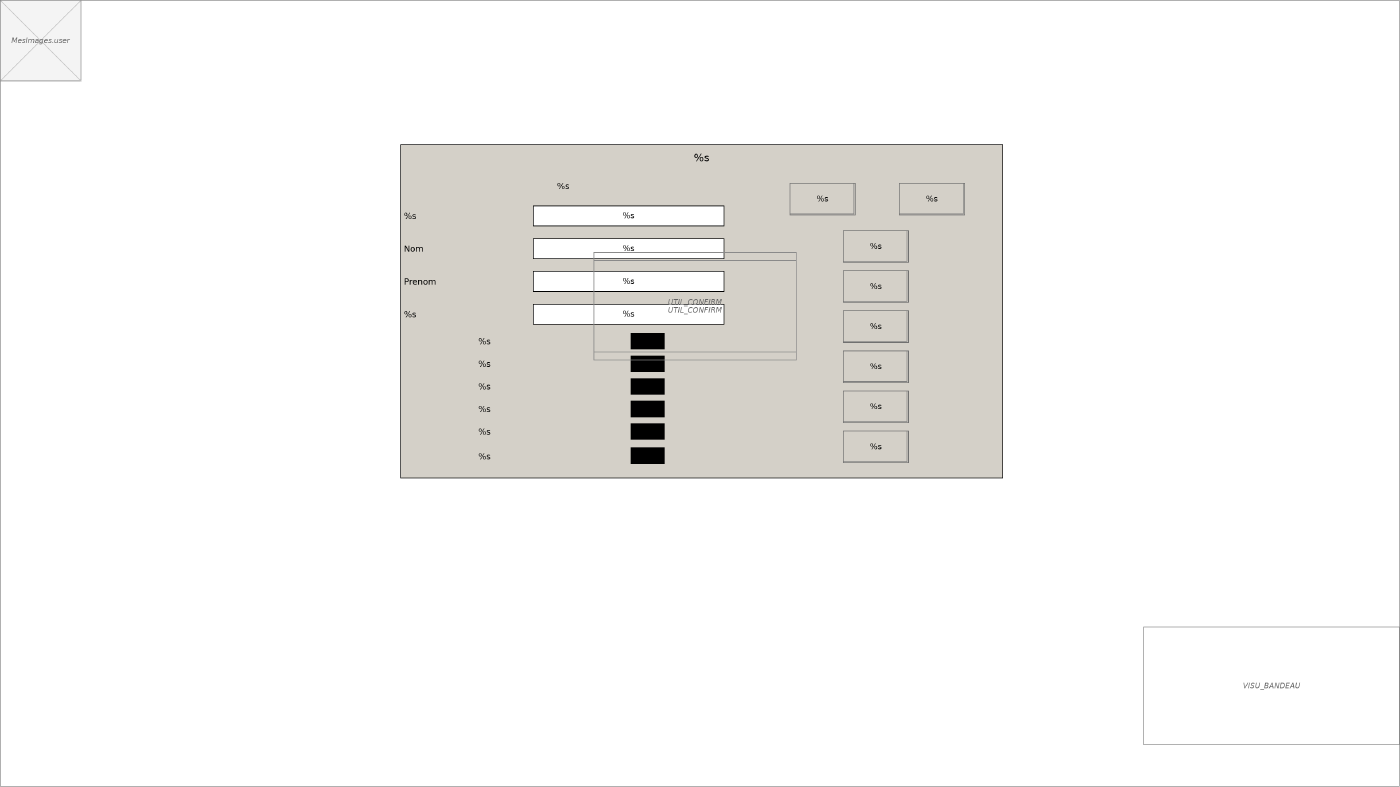
VISUALIZATION UTIL_MENU  // 1920x1080
    Image (0,0 111x111), image: MesImages.user
    RoundedRectangle (549,198 826x458)
    Rectangle (553,202 819x29), "%s", text list: 'TextList_Users_Menu', text index: 1
    Rectangle (731,282 262x28), "%s", text variable: PRG_USER.ACTU_USER.LOGIN
    Rectangle (552,241 441x29), "%s", text list: 'TextList_Users_Menu', text index: 7
    Rectangle (551,282 173x29), "%s", text list: 'TextList_Users_Menu', text index: 5
    Rectangle (551,327 173x29), "Nom"
    Rectangle (551,372 173x29), "Prenom"
    Rectangle (731,327 262x28), "%s", text variable: PRG_USER.ACTU_USER.NOM
    Rectangle (731,372 262x28), "%s", text variable: PRG_USER.ACTU_USER.PRENOM
    Rectangle (551,417 173x29), "%s", text list: 'TextList_Users_Menu', text index: 8
    Rectangle (731,417 262x28), "%s", text variable: PRG_USER.ACTU_USER.GROUPE
        OnMouseClick: write the text variable via VisuDialogs.Keypad
    Rectangle (653,485 112x29), "%s", text list: 'TextList_Util_Group', text index: 4
    Rectangle (653,516 112x29), "%s", text list: 'TextList_Util_Group', text index: 5
    Rectangle (653,454 112x29), "%s", text list: 'TextList_Util_Group', text index: 3
    Rectangle (653,547 112x29), "%s", text list: 'TextList_Util_Group', text index: 6
    Rectangle (653,578 112x29), "%s", text list: 'TextList_Util_Group', text index: 7
    Rectangle (653,612 122x29), "%s", text list: 'TextList_Util_Group', text index: 8
    Rectangle (865,457 46x22), "Oui", colour toggle: PRG_USER.ACTU_USER.PROGRAMMATION
    Rectangle (865,488 46x22), "Oui", colour toggle: PRG_USER.ACTU_USER.MAINTENANCE
    Rectangle (865,519 46x22), "Oui", colour toggle: PRG_USER.ACTU_USER.SUPERVISEUR
    Rectangle (865,550 46x22), "Oui", colour toggle: PRG_USER.ACTU_USER.PRODUCTION
    Rectangle (865,581 46x22), "Oui", colour toggle: PRG_USER.ACTU_USER.CONF_MACHINE
    Rectangle (865,614 46x22), "Oui", colour toggle: PRG_USER.ACTU_USER.FONCTION_SA
    Button (1083,251 90x44), "%s", input disabled if: PRG_USER.UTIL_EC, text list: 'TextList_Users_Menu', text index: 9
        toggle PRG_USER.DD_LOG1
        OnMouseClick: change screen: UTIL_LOG
    Button (1233,251 90x44), "%s", input disabled if: MAIN.VAR_INVISIBLE_DELOG, text list: 'TextList_Users_Menu', text index: 10
        OnMouseClick: change screen: UTIL_DELOG
    Button (1156,316 90x44), "%s", input disabled if: NOT PRG_USER.ACTU_USER.SUPERVISEUR, text list: 'TextList_Users_Menu', text index: 11
        toggle PRG_USER.DD_mod_def1
        OnMouseClick: change screen: UTIL_DEFAUT
    Button (1156,371 90x44), "%s", input disabled if: NOT PRG_USER.ACTU_USER.SUPERVISEUR, text list: 'TextList_Users_Menu', text index: 12
        OnMouseClick: change screen: UTIL_USER
    Button (1156,426 90x44), "%s", input disabled if: NOT PRG_USER.ACTU_USER.SUPERVISEUR, text list: 'TextList_Users_Menu', text index: 13
        OnMouseClick: change screen: UTIL_GROUP
    Button (1156,481 90x44), "%s", input disabled if: PRG_USER.LOAD_EC OR NOT PRG_USER.ACTU_USER.SUPERVISEUR OR PRG_USER.SAVE_EC, text list: 'TextList_Users_Menu', text index: 14
        toggle PRG_USER.VISU_FEN1
    Button (1156,536 90x44), "%s", input disabled if: PRG_User.SAVE_EC OR NOT PRG_User.ACTU_USER.SUPERVISEUR OR PRG_User.LOAD_EC, text list: 'TextList_Users_Menu', text index: 15
        toggle PRG_USER.VISU_FEN2
    Button (1156,591 90x44), "%s", input disabled if: NOT PRG_USER.ACTU_USER.SUPERVISEUR, text list: 'TextList_Users_Menu', text index: 16
        toggle PRG_USER.DD_mod_def1
        OnMouseClick: change screen: UTIL_OPT
    Frame (814,346 278x137), invisible if: NOT PRG_USER.VISU_FEN1
        shows UTIL_CONFIRM(Num_Text := 20, OrdreDD := PRG_USER.DD_load, Visu := PRG_USER.VISU_FEN1)
    Frame (814,357 278x137), invisible if: NOT PRG_USER.VISU_FEN2
        shows UTIL_CONFIRM(Num_Text := 17, OrdreDD := PRG_USER.DD_sauv, Visu := PRG_USER.VISU_FEN2)
    Frame (1568,860 352x162)
        shows VISU_BANDEAU(m_Input_MACHINE := Global_Variables.MACHINE)
END_VISUALIZATION

(* stored: Version 1.1.0.1, ProductVersion 3.1.4024.10
   Visu UTIL_MENU: Id {ee2f8c70-4681-4407-88bf-aef42da37d42} *)
